TYPE READ_ADS_EVENT_DATA :
STRUCT
	Class			: E_TcEventClass;
	id				: DWORD;
	State			: DWORD;
	Question		: DWORD;
	SourceId		: DWORD;
	Source			: STRING(80);
	DateAndTime		: DT;
	Computer		: STRING(80);
	MsgText			: STRING(500);
END_STRUCT
END_TYPE

(* stored: Version 1.1.0.1, ProductVersion 3.1.4024.12
   DUT READ_ADS_EVENT_DATA: Id {72ffa2b3-3569-40bd-b45a-2fe5642d21b7} *)
